INTERFACE I_CalcThicknessFromXRayTransmission EXTENDS I_Fallible


METHOD Calculate
VAR_INPUT
    MaterialFormula : T_MaxString;
    Transmission : I_QuantityLREAL;
    Thickness : I_QuantityLREALPublic;
END_VAR
END_METHOD

END_INTERFACE

(* stored: Version 1.1.0.1
   Itf I_CalcThicknessFromXRayTransmission: Id {7392466d-a1ca-4218-bf3e-e96dfd30823e}
   Method Calculate: Id {dbdd9771-bb12-49af-8778-a0e433a83d02} *)
